# B&R Automation Studio project ABC_Pltzr (part 2)

#### bgTcpSocketClient.c
```c
/*
File: bgTcpSocketClientServer.c
=====

B&R Libraries:
==============
Make sure to add following .a files to the task using this source file:
libsys_lib.a
libbrsystem.a
libastcp.a
*/

/*
B&R components:
===============================================================================
*/
#include <bur/plc.h>
#include <bur/plctypes.h>
#include <ethsock.h>
#include <astcp.h>
#include <brsystem.h>
#include <sys_lib.h>

/*
BG components
===============================================================================
*/
#include "bgdebug.h"
#include "bgstring.h"

#include "bgTcpSocketClientServer.h"
#include "bgHttpProtocol.h"

/*
Tcp Socket Client
*/
static void bgTcpSocketClientDefaultSessionHandler(bgTcpSocketSession_typ* pSession);
static void bgTcpSocketClientSessionStateMachine(bgTcpSocketSession_typ* pSession);
static void	bgTcpSocketClientExecuteSessionHandler(bgTcpSocketSession_typ* pSession, int init);

static void bgTcpSocketClientMemAlloc(bgTcpSocketClient_typ* pClient);
static void bgTcpSocketClientSessionStart(bgTcpSocketClient_typ* pClient);
static void	bgTcpSocketClientExecuteSessionHandler(bgTcpSocketSession_typ* pSession, int init);
static void bgTcpSocketClientSessionCyclic(bgTcpSocketClient_typ* pClient);
static void bgTcpSocketClientSessionLauncher(bgTcpSocketClient_typ* pClient);
static void setSocketAddressData(ETH_sockaddr_typ *adrData, char *hostIpAddressString, unsigned short hostPort);
static void swapBytesInShort(unsigned short *value);

/*
TCP Socket Client
######################################################################################################
######################################################################################################
######################################################################################################
######################################################################################################
*/
void bgTcpSocketClientInit(bgTcpSocketClient_typ* pClient,
    int sessionSendBufSize,
    int sessionRecvBufSize,
    int applicationBufSize,
    char* pRecvBuf,
    void (*pSessionHandler)(bgTcpSocketSession_typ*),
    void (*pApplicationHandler)(bgTcpSocketSession_typ*))
{
    pClient->serverPort = 0;

	pClient->recvBuffer = pRecvBuf;

	/*Recv buffer can't be allocated! recv DOES NOT WORK if the buffer is not in PV space!?!?!?!?*/
	if(!pRecvBuf){
		DBGCRT("bgTcpSocketClientInit: recvBuf not defined!\r\n");
		pClient->memAllocStatus2 = 1;
		return;
	}

    pClient->serverIpAddr[0] = 0;

    pClient->numSupportedSessions = 1;

    pClient->sessionSendBufSize = sessionSendBufSize;

    pClient->sessionRecvBufSize = sessionRecvBufSize;

	pClient->applicationBufSize = applicationBufSize;

	/*Recv buffer can't be allocated! recv DOES NOT WORK if the buffer is not in PV space!?!?!?!?*/
    pClient->sessionTotalBufSize = pClient->sessionSendBufSize + pClient->applicationBufSize;

    pClient->totalBufSize = pClient->sessionTotalBufSize * pClient->numSupportedSessions;

    pClient->pSessionHandler = pSessionHandler;

    pClient->pApplicationHandler = pApplicationHandler;

	pClient->sockStateData = BGTCPSOCK_STATE_NONE;

	pClient->dbgDumpSendBuf = 0;
	pClient->dbgDumpRecvBuf = 0;

	/*allocate memory for send/recv buffers*/
	bgTcpSocketClientMemAlloc(pClient);

	if(pClient->memAllocStatus2 ){
			DBGCRT("bgTcpSocketClientInit: memory error! memAllocStatus2=%d\r\n", pClient->memAllocStatus2);
	}
}

void bgTcpSocketClientCyclic(bgTcpSocketClient_typ* pClient)
{
int ret;
	/*non-blocking I/O control*/
static ETH_fd_set_typ fdR;
static ETH_fd_set_typ fdW;
static ETH_timeval_typ timeOut;

	/*if memalloc fails, can't do much!*/
	if(pClient->memAllocStatus2)
		return;

	/*monitor upper layer requests to start a client session*/
	bgTcpSocketClientSessionLauncher(pClient);

	/*execute session state machine*/
	bgTcpSocketClientSessionCyclic(pClient);

	/*client state machine*/
	switch(pClient->sockStateData){
		case BGTCPSOCK_STATE_NONE:
    		return;
		break;

		case BGTCPSOCK_STATE_INITOPEN:

 			/*create socket*/
			pClient->tcpOpen.ident = socket(ETH_AF_INET, ETH_SOCK_STREAM, 0);

			if( pClient->tcpOpen.ident == ERR_SOCKET ){
				DBGMSG("socket create error (init open); EthGetError=%d\r\n", EthGetError());
				pClient->sockStateData = BGTCPSOCK_STATE_NONE;
				break;
			}

			pClient->tcpClient.ident = pClient->tcpOpen.ident;
			pClient->tcpClose.ident = pClient->tcpOpen.ident;

			/*set non-blocking socket operation*/
			{
				UDINT arg = 1;
				ioctl(pClient->tcpOpen.ident, ETH_FIONBIO, (UDINT)&arg);
			}

#if 0
			/*get sock options*/
			{
				ret = getsockopt(pClient->tcpOpen.ident, ETH_SOL_SOCKET, ETH_SO_SNDTIMEO, (UDINT)&opt1, (UDINT)&opt1size);
				DBGMSG("getsockopt ret=%d\r\n", ret);
			}
#endif

			/*reset select flags*/
			fd_zero((UDINT)&fdR);
			fd_zero((UDINT)&fdW);

			/*set time-out to 10ms*/
			timeOut.tv_sec = 0;
			timeOut.tv_usec = 1000 * 10;

			pClient->sockStateData = BGTCPSOCK_STATE_OPEN;

		case BGTCPSOCK_STATE_OPEN:

			/*connect to remote host*/
			{
			ETH_sockaddr_typ serverAdr;
			setSocketAddressData(&serverAdr, pClient->serverIpAddr, pClient->serverPort);
			ret = connect(pClient->tcpOpen.ident, (UDINT)&serverAdr, sizeof(ETH_sockaddr_typ) );
			}

			if(ret == ERR_SOCKET){
				UINT errCode = EthGetError();
				if(errCode == ERR_ETH_INPROGRESS){
					/*next: wait connect to complete*/
					DBGMSG("socket connect - wait connect to complete!\r\n");
					pClient->sockStateData = BGTCPSOCK_STATE_CLIENT;
				    break;
				}else
				if(errCode == ERR_ETH_ISCONN){
					/*it's connected -> done*/
					DBGMSG("socket connect ok(1)!\r\n");
	                bgTcpSocketClientSessionStart(pClient);
					pClient->sockStateData = BGTCPSOCK_STATE_CONNECTED;
					break;
				}
				else{
					DBGMSG("socket connect error(open); EthGetError=%d\r\n", EthGetError());
					pClient->sockStateData = BGTCPSOCK_STATE_NONE;
					break;
				}
			}
			/*connected!*/
			/*it's connected -> done*/
			DBGMSG("socket connect ok(2)!\r\n");
            bgTcpSocketClientSessionStart(pClient);
			pClient->sockStateData = BGTCPSOCK_STATE_CONNECTED;
		break;
		case BGTCPSOCK_STATE_CLIENT:
			/*select waits for connection to complete*/
			fd_set(pClient->tcpOpen.ident, (UDINT)&fdR);
			fd_set(pClient->tcpOpen.ident, (UDINT)&fdW);
			ret = sock_select(32, (UDINT)&fdR, (UDINT)&fdW, 0L, (UDINT)&timeOut);

			if(ret == ERR_SOCKET){
				DBGMSG("socket connect error; (cli) EthGetError=%d\r\n", EthGetError());
				pClient->sockStateData = BGTCPSOCK_STATE_CLOSE;
				break;
			}

			if(ret == 0){

			}else{
				if( fd_isset(pClient->tcpOpen.ident, (UDINT)&fdW) ){
					DBGMSG("socket connect(long) ok!\r\n");
	                bgTcpSocketClientSessionStart(pClient);
					pClient->sockStateData = BGTCPSOCK_STATE_CONNECTED;
				}
			}
		break;
        case BGTCPSOCK_STATE_CONNECTED:
			/*Monitor session operation; generate OnResponseReady & OnResponseError triggers*/
            /*TODO: implement timeout here -> kill sessions if stuck*/
			if(pClient->session[0].socketState == BGTCPSOCK_SESSION_STATE_NONE){
				pClient->sockStateData = BGTCPSOCK_STATE_NONE;
			}
        break;
        case BGTCPSOCK_STATE_CLOSE:
			close(pClient->tcpClose.ident);
	    	pClient->sockStateData = BGTCPSOCK_STATE_NONE;
			DBGMSG("bgTcpSocketClientSessionStateMachine(): closing socket\r\n");
        break;
        case BGTCPSOCK_STATE_ERROR:
        break;
	 }

    return;
}

static void bgTcpSocketClientMemAlloc(bgTcpSocketClient_typ* pClient)
{
unsigned int memSize;
int i;

	/*Get System Memory Information*/
	pClient->MEMInfo.enable = 1;
	MEMInfo(&pClient->MEMInfo);

	memSize = pClient->totalBufSize;

	/*allocate space for send/recv buffers*/
	if(pClient->sendRecvBuffer == 0){
		/* allocate new memory from RAM*/
    	pClient->memAllocStatus2 = TMP_alloc(memSize, (void**)&pClient->sendRecvBuffer);
	}else{
		/*memory is allready allocated -> free it first!*/
    	pClient->memAllocStatus2 = TMP_free(memSize, (void**)pClient->sendRecvBuffer);

    	/*allocate new memory from RAM*/
    	pClient->memAllocStatus2 = TMP_alloc(memSize, (void**)pClient->sendRecvBuffer);
	}

	/*assign send/recv buffer ptrs*/
    pClient->session[0].pSendBuf = (char*)(pClient->sendRecvBuffer + i * pClient->sessionTotalBufSize);
	pClient->session[0].sendBufLength = pClient->sessionSendBufSize;

    pClient->session[0].pAppBuf = (char*)(pClient->session[0].pSendBuf + pClient->sessionSendBufSize);
	pClient->session[0].appBufLength = pClient->applicationBufSize;

    pClient->session[0].pRecvBuf = pClient->recvBuffer;
	pClient->session[0].recvBufLength = pClient->sessionRecvBufSize;
}

static void bgTcpSocketClientSessionStart(bgTcpSocketClient_typ* pClient)
{
int i;
bgTcpSocketSession_typ *pSession;

	/* client: pClient->numSupportedSessions = 1 ALWAYS!*/
    for(i=0; i < pClient->numSupportedSessions; i++){
        if( pClient->session[i].socketState == BGTCPSOCK_SESSION_STATE_NONE){
            pSession = &pClient->session[i];
            pSession->socketState = BGTCPSOCK_SESSION_STATE_SEND;

			pSession->tcpSend.enable = 1;
			pSession->tcpSend.ident = pClient->tcpOpen.ident;   		/* copy the  Ident number */
			pSession->tcpSend.flags = 0;
			pSession->tcpSend.pData = (UDINT)pSession->pSendBuf;

			pSession->tcpRecv.enable = 1;
			pSession->tcpRecv.ident = pClient->tcpOpen.ident;     		/* copy the  Ident number */

			pSession->tcpRecv.pData = (UDINT)pSession->pRecvBuf;        /* address of the buffer */;

			pSession->tcpRecv.datamax = pClient->sessionRecvBufSize;    /* length of the buffer */;

			pSession->tcpClose.enable = 1;
   			pSession->tcpClose.ident = pClient->tcpOpen.ident;    		/* copy the  Ident number */

			pSession->pTcpLayer = (char*)pClient;	                    /*session has ptr to tcp layer*/

            pSession->rxByteCount = 0;
            brsstrcpy((UDINT)pSession->clientIpAddr, (UDINT)pClient->clientIpAddr);

			pSession->dbgDumpRecvBuf = pClient->dbgDumpRecvBuf;
			pSession->dbgDumpSendBuf = pClient->dbgDumpSendBuf;

			/*init session specific handler - call the handler with init pSession->flag=1*/
			bgTcpSocketClientExecuteSessionHandler(pSession, 1);

			DBGMSG("bgTcpSocketClientSessionStart(): connection to %s, starting session Id= %d\r\n", pClient->serverIpAddr, i);
            return;
        }
    }

	DBGCRT("bgTcpSocketClientSessionStart(): client busy! activeSessions= %d\r\n", pClient->numSupportedSessions);
    pClient->sockStateData = BGTCPSOCK_STATE_TOOBUSY;
}

static void	bgTcpSocketClientExecuteSessionHandler(bgTcpSocketSession_typ* pSession, int init)
{
bgTcpSocketClient_typ* pClient = (bgTcpSocketClient_typ*)pSession->pTcpLayer;

	pSession->init = 0;
	if( init )
		pSession->init = 1;

	DBGMSG("bgTcpSocketClientExecuteSessionHandler\r\n p1=%d p2=%d\r\n", pClient->pSessionHandler, bgHttpClientSessionHandler);

/*
	bgHttpClientSessionHandler(pSession);
*/
    if(pClient->pSessionHandler)
    	(*pClient->pSessionHandler)(pSession);
    else
    	bgTcpSocketClientDefaultSessionHandler(pSession);

	pSession->init = 0;
}

static void bgTcpSocketClientSessionCyclic(bgTcpSocketClient_typ* pClient)
{
int i;
bgTcpSocketSession_typ *pSession;
int activeSessions = 0;

    for(i=0; i < pClient->numSupportedSessions; i++){
        pSession = &pClient->session[i];

        if( pSession->socketState != BGTCPSOCK_SESSION_STATE_NONE){
            activeSessions++;
            bgTcpSocketClientSessionStateMachine(pSession);
        }
    }
    pClient->numActiveSessions = activeSessions;
}

static void bgTcpSocketClientSessionLauncher(bgTcpSocketClient_typ* pClient)
{
int i;
bgTcpSocketSession_typ *pSession;

    for(i=0; i < pClient->numSupportedSessions; i++){
        pSession = &pClient->session[i];

		if( (pSession->bSendData) ){
			pSession->bSendData = 0;
			if(pClient->sockStateData == BGTCPSOCK_STATE_NONE){
				pClient->sockStateData = BGTCPSOCK_STATE_INITOPEN;
			}else{
				DBGMSG("bgTcpSocketClientSessionLauncher: client session start rejected; client is busy! cliState=%d\r\n",
					pClient->sockStateData);
			}
		}
    }
}
static void bgTcpSocketClientSessionStateMachine(bgTcpSocketSession_typ* pSession)
{
int ret;

    switch(pSession->socketState){
		case BGTCPSOCK_SESSION_STATE_SEND:

        	ret = send(pSession->tcpSend.ident, (UDINT)pSession->pSendBuf, pSession->tcpSend.datalen, 0L);

        	if(ret == ERR_SOCKET){
				DBGMSG("send error EthGetError=%d\r\n", EthGetError());
				pSession->socketState = BGTCPSOCK_SESSION_STATE_CLOSE;    /*close this socket*/
				return;
        	}

			/*remember the send length*/
			DBG("send() ok; bytes=%d\r\n", (int)ret);
			pSession->tcpSend.sentlen = ret;
	   		pSession->socketState = BGTCPSOCK_SESSION_STATE_RECEIVE;    /*close this socket session*/

		/*break;*/

		case BGTCPSOCK_SESSION_STATE_RECEIVE:
	       	/*call receive (NON BLOCKING MODE!)*/
        	ret = recv(pSession->tcpRecv.ident, (UDINT)pSession->tcpRecv.pData, pSession->tcpRecv.datamax, 0L);

        	if(ret == ERR_SOCKET){
        		UINT errCode = EthGetError();
        		/*none blocking receive return this following value if data is not available yet*/
        		if( errCode == ERR_ETH_WOULDBLOCK ){
        			/*wait response*/
					return;
        		}
				DBGMSG("RxError EthGetError=%d\r\n", errCode);
	   			pSession->socketState = BGTCPSOCK_SESSION_STATE_CLOSE;    /*close this socket session*/
				break;
        	}

			pSession->tcpRecv.recvlen = ret;

            if(pSession->tcpRecv.recvlen){
				DBGMSG("rx OK! rxLen=%d\r\n", ret);

				bgTcpSocketClientExecuteSessionHandler(pSession, 0);

				/*uper layer completed processing? */
				if( pSession->bCloseSession){
					pSession->bCloseSession = 0;
	   					pSession->socketState = BGTCPSOCK_SESSION_STATE_CLOSE;    /*close this socket session*/
				}
            }else{
				DBGMSG("bgTcpSocketClient..: RMT SOCK CLOSED!\r\n");
	   			pSession->socketState = BGTCPSOCK_SESSION_STATE_CLOSE;    /*close this socket session*/
			}
			return;
		break;

		case BGTCPSOCK_SESSION_STATE_CLOSE:
			close(pSession->tcpClose.ident);
	    	pSession->socketState = BGTCPSOCK_SESSION_STATE_NONE;
			DBGMSG("bgTcpSocketClientSessionStateMachine(): stopping session Id= %d\r\n", pSession->ident);
		break;

		case BGTCPSOCK_SESSION_STATE_DELAY:
			pSession->delayCounter--;
			if(pSession->delayCounter <= 0)
    			pSession->socketState = BGTCPSOCK_SESSION_STATE_CLOSE;    /*close this server socket*/
		break;

		default:

		break;
	}
}

#if 0
static void bgTcpSocketClientSessionSendData(bgTcpSocketSession_typ* pSession, int len)
{
	pSession->tcpSend.datalen = len;
	pSession->socketState = BGTCPSOCK_STATE_INITOPEN;

#if 0
{
int i;
char text[90];
/*session/application/protocol specific data structure*/
httpRequest_typ* r = (httpRequest_typ*)pSession->pProtocol;

	DBGMSG("bgHttpSend(): lenght(bytes): total=%d(%d) header=%d content=%d\r\n",
		len, r->sendTotalLength, r->sendHeaderLength, r->sendContentLength);

	DBGMSG("bgHttpSend dump:\r\n");
	DBGMSG("============================================\r\n");
	for(i=0;i<len; i++){
 		if( ((i+1)*80) < len ){
			memcpy(&text[0], &pSession->pSendBuf[i*80], 80);
			text[80]=0;
			DBGMSG("%s", &text[0]);
		}else{
			memcpy(&text[0], &pSession->pSendBuf[i*80], len - (i*80));
			text[len - (i*80)]=0;
			DBGMSG("%s", &text[0]);
			break;
		}
	}
	DBGMSG("============================================\r\n\r\n");
}
#endif

}
#endif
/*
Default session handler
######################################################################################################
######################################################################################################
######################################################################################################
######################################################################################################
*/
static void bgTcpSocketClientDefaultSessionHandler(bgTcpSocketSession_typ* pSession)
{
    /*default session handler -> send out http error response "internal server error"*/
/*    httpSendErrorResponse(pSession, 500);
*/
}

static void setSocketAddressData(ETH_sockaddr_typ *adrData, char *hostIpAddressString, unsigned short hostPort)
{

	unsigned short sin_family;
	unsigned short family;
	unsigned short length;
	unsigned short port;

	family = ETH_AF_INET;
	length = sizeof(ETH_sockaddr_typ);
	sin_family = (family << 8) + length;

	adrData->sin_family = sin_family;
	port = hostPort;
	swapBytesInShort(&port);
	adrData->sin_port = port;
	if( strlen(hostIpAddressString) < 8)
		adrData->sin_addr = ETH_INADDR_ANY;
	else
		adrData->sin_addr = inet_addr( (unsigned long) hostIpAddressString);
	adrData->sin_zero[0]=0;
	adrData->sin_zero[1]=0;
	adrData->sin_zero[2]=0;
	adrData->sin_zero[3]=0;
	adrData->sin_zero[4]=0;
	adrData->sin_zero[5]=0;
	adrData->sin_zero[6]=0;
	adrData->sin_zero[7]=0;
}

static void swapBytesInShort(unsigned short *value)
{

union{
	unsigned short 	shortValue;
	unsigned char	bytes[2];
}swapValue;

unsigned char tempByte;

	swapValue.shortValue = *value;
	tempByte = swapValue.bytes[0];
	swapValue.bytes[0] = swapValue.bytes[1];
	swapValue.bytes[1] = tempByte;
	*value = swapValue.shortValue;
}
```

### paiFileService.typ
```iecst
(********************************************************************
 * COPYRIGHT --
 ********************************************************************
 * Package: paiFileService
 * File: paiFileService.typ
 * Author: goran_2
 * Created: August 05, 2011
 ********************************************************************
 * Data types of package paiFileService
 ********************************************************************)

TYPE
	PAI_FILESERVICE_ENUMS :
		(
		PAI_FS_DEVICE_MAXIDX := 19,
		PAI_FS_DEVICE_NONE := 0,
		PAI_FS_IDLE := 0,
		PAI_FS_RDFILE := 1,
		PAI_FS_WRFILE := 2,
		PAI_FS_INFOFILE := 3,
		PAI_FS_DELFILE := 4,
		PAI_FS_RDDIR := 10,
		PAI_FS_CRDIR := 11,
		PAI_FS_INFODIR := 12
		);
	paiFileServiceDevDirItem_typ : 	STRUCT
		deviceName : STRING[31];
		dirName : STRING[127];
		deviceConfiguration : STRING[127];
		createdAtPowerUp : BOOL;
		status : INT;
	END_STRUCT;
	paiFileServiceDeviceTable_typ : 	STRUCT
		listDevsDirs : ARRAY[0..19]OF paiFileServiceDevDirItem_typ;
	END_STRUCT;
	paiFileServicePublicIn_typ : 	STRUCT
		request : USINT;
		adrDeviceName : UDINT; (*Address of the Device Name*)
		adrName : UDINT; (*File/dir name for the requested action (read, write, create, delete, etc)*)
		adrName2 : UDINT; (*File/dir name for the requested action (read, write, create, delete, etc)*)
		adrReadDst : UDINT; (*Destination address for the read action*)
		readDstLen : UDINT; (*Length of the space available for read at the given address*)
		readOffset : UDINT;
		adrWriteSrc : UDINT; (*Src address for the write action.*)
		writeSrcLen : UDINT; (*Length of data available at src address*)
		writeOffset : UDINT;
		pCallback : UDINT; (*ptr to Callback function*)
		pCallbackData : UDINT; (*ptr to Callback data*)
	END_STRUCT;
	paiFileServicePublicOut_typ : 	STRUCT
		status : UINT; (*Output status for R or W request. Valid when writeDone or readDone set to 1.*)
		initOk : BOOL; (*Output status that indicates if service completed initialization after system start. Wait with any access until initOk == 1*)
		busy : BOOL; (*Output status to indicate that service is busy (busy == 1) servicing a current request. Avoid issuing new requests.*)
		powerUp : BOOL; (*Output status to indicate that service completed servicing a current request. Shall be cleared by the receiver of the event.*)
		done : BOOL; (*Output status to indicate that service completed servicing a current request. Shall be cleared by the receiver of the event.*)
		bytecount : UDINT; (*Number of bytes during file read.*)
	END_STRUCT;
	paiFileServicePrivateFileFBK_typ : 	STRUCT
		open : FileOpen;
		close : FileClose;
		read : FileRead;
		readex : FileReadEx;
		write : FileWrite;
		writeex : FileWriteEx;
		copy : FileCopy;
		create : FileCreate;
		delete : FileDelete;
		rename : FileRename;
		truncate : FileTruncate;
		info : FileInfo;
		infoData : fiFILE_INFO;
	END_STRUCT;
	paiFileServicePrivateDevFBK_typ : 	STRUCT
		link : DevLink;
		unlink : DevUnlink;
	END_STRUCT;
	paiFileServiceDirFBK_typ : 	STRUCT
		open : DirOpen;
		close : DirClose;
		read : DirRead;
		copy : DirCopy;
		create : DirCreate;
		delete : DirDelete;
		deleteex : DirDeleteEx;
		rename : DirRename;
		info : DirInfo;
	END_STRUCT;
	paiFileServicePrivate_typ : 	STRUCT
		requestType : USINT;
		status : UINT;
		bgssm : bgSSM_typ;
		currentDeviceIndex : UDINT;
		pDeviceTable : REFERENCE TO paiFileServiceDeviceTable_typ;
		device : paiFileServicePrivateDevFBK_typ;
		dir : paiFileServiceDirFBK_typ;
		file : paiFileServicePrivateFileFBK_typ;
	END_STRUCT;
	paiFileService_typ : 	STRUCT
		i : paiFileServicePublicIn_typ;
		o : paiFileServicePublicOut_typ;
		prv : paiFileServicePrivate_typ;
	END_STRUCT;
END_TYPE
```

### Program Logical/paiComponents/paiFileService/paiFS (ANSIC)

#### paiDevDirConfigure.c - pai FS Device and Directory configuration
```c
/********************************************************************
 * COPYRIGHT --
 ********************************************************************
 * Program: paiFile
 * File: paiDevDirConfigure.c
 * Author: goran_2
 * Created: August 05, 2011
 ********************************************************************
 * Implementation of program paiDevDirConfigure
 ********************************************************************/

#include <bur/plctypes.h>

#ifdef _DEFAULT_INCLUDES
 #include <AsDefault.h>
#endif

#include "paiFile.h"

/*
###############################################################################
PAI_CONFIGURATION_SECTION
Code below allows configuration of the devices and folders used in the
application.
###############################################################################
*/
#warning "pai Configuration: application File Devices and Folders"
void paiFSDeviceAndDirConfig( void )
{
	int idx=0;
	//If .deviceConfiguration is NOT empty string, entry is related to device link at powerup
	//If .deviceConfiguration is empty string, entry is related to directory check/create at powerup

	brsstrcpy((UDINT)paiFSDevices.listDevsDirs[idx].deviceName, (UDINT)PAI_FS_DEVICE_ROOT);
	brsstrcpy((UDINT)paiFSDevices.listDevsDirs[idx].dirName, (UDINT)"");
	brsstrcpy((UDINT)paiFSDevices.listDevsDirs[idx].deviceConfiguration, (UDINT)PAI_FS_DEVICE_ROOT_CFG);

	idx++;
	brsstrcpy((UDINT)paiFSDevices.listDevsDirs[idx].deviceName, (UDINT)PAI_FS_DEVICE_ROOT);
	brsstrcpy((UDINT)paiFSDevices.listDevsDirs[idx].dirName, (UDINT)PAI_FS_APP_DIR_DATA);//i.e. Data
	brsstrcpy((UDINT)paiFSDevices.listDevsDirs[idx].deviceConfiguration, (UDINT)"");

	idx++;
	brsstrcpy((UDINT)paiFSDevices.listDevsDirs[idx].deviceName, (UDINT)PAI_FS_DEVICE_ROOT);
	brsstrcpy((UDINT)paiFSDevices.listDevsDirs[idx].dirName, (UDINT)PAI_FS_APP_DIR_CFG);//i.e. Data/Cfg
	brsstrcpy((UDINT)paiFSDevices.listDevsDirs[idx].deviceConfiguration, (UDINT)"");

	idx++;
	brsstrcpy((UDINT)paiFSDevices.listDevsDirs[idx].deviceName, (UDINT)PAI_FS_DEVICE_ROOT);
	brsstrcpy((UDINT)paiFSDevices.listDevsDirs[idx].dirName, (UDINT)PAI_FS_APP_DIR_REC);//i.e. Data/Rec
	brsstrcpy((UDINT)paiFSDevices.listDevsDirs[idx].deviceConfiguration, (UDINT)"");

	idx++;
	brsstrcpy((UDINT)paiFSDevices.listDevsDirs[idx].deviceName, (UDINT)PAI_FS_DEVICE_ROOT);
	brsstrcpy((UDINT)paiFSDevices.listDevsDirs[idx].dirName, (UDINT)"Data/Rec/Layers");//i.e. Data/Rec/Layers
	brsstrcpy((UDINT)paiFSDevices.listDevsDirs[idx].deviceConfiguration, (UDINT)"");

	idx++;
	brsstrcpy((UDINT)paiFSDevices.listDevsDirs[idx].deviceName, (UDINT)PAI_FS_DEVICE_ROOT);
	brsstrcpy((UDINT)paiFSDevices.listDevsDirs[idx].dirName, (UDINT)"Data/Rec/Pallets");//i.e. Data/Rec/Pallets
	brsstrcpy((UDINT)paiFSDevices.listDevsDirs[idx].deviceConfiguration, (UDINT)"");

	idx++;
	brsstrcpy((UDINT)paiFSDevices.listDevsDirs[idx].deviceName, (UDINT)PAI_FS_DEVICE_ROOT);
	brsstrcpy((UDINT)paiFSDevices.listDevsDirs[idx].dirName, (UDINT)"Data/Test");
	brsstrcpy((UDINT)paiFSDevices.listDevsDirs[idx].deviceConfiguration, (UDINT)"");

	idx++;
	brsstrcpy((UDINT)paiFSDevices.listDevsDirs[idx].deviceName, (UDINT)PAI_FS_DEVICE_CFG);
	brsstrcpy((UDINT)paiFSDevices.listDevsDirs[idx].dirName, (UDINT)"");
	brsstrcpy((UDINT)paiFSDevices.listDevsDirs[idx].deviceConfiguration, (UDINT)PAI_FS_DEVICE_CFG_CFG);

	idx++;
	brsstrcpy((UDINT)paiFSDevices.listDevsDirs[idx].deviceName, (UDINT)PAI_FS_DEVICE_REC);
	brsstrcpy((UDINT)paiFSDevices.listDevsDirs[idx].dirName, (UDINT)"");
	brsstrcpy((UDINT)paiFSDevices.listDevsDirs[idx].deviceConfiguration, (UDINT)PAI_FS_DEVICE_REC_CFG);

	idx++;
	brsstrcpy((UDINT)paiFSDevices.listDevsDirs[idx].deviceName, (UDINT)PAI_FS_DEVICE_REC_LAYER);
	brsstrcpy((UDINT)paiFSDevices.listDevsDirs[idx].dirName, (UDINT)"");
	brsstrcpy((UDINT)paiFSDevices.listDevsDirs[idx].deviceConfiguration, (UDINT)PAI_FS_DEVICE_REC_LAYER_CFG);

	idx++;
	brsstrcpy((UDINT)paiFSDevices.listDevsDirs[idx].deviceName, (UDINT)PAI_FS_DEVICE_REC_PALLETE);
	brsstrcpy((UDINT)paiFSDevices.listDevsDirs[idx].dirName, (UDINT)"");
	brsstrcpy((UDINT)paiFSDevices.listDevsDirs[idx].deviceConfiguration, (UDINT)PAI_FS_DEVICE_REC_PALLETE_CFG);

	idx++;
	brsstrcpy((UDINT)paiFSDevices.listDevsDirs[idx].deviceName, (UDINT)"USB1");
	brsstrcpy((UDINT)paiFSDevices.listDevsDirs[idx].dirName, (UDINT)"");
	brsstrcpy((UDINT)paiFSDevices.listDevsDirs[idx].deviceConfiguration, (UDINT)"/DEVICE=IF3.ST1");

	idx++;
	brsstrcpy((UDINT)paiFSDevices.listDevsDirs[idx].deviceName, (UDINT)"USB2");
	brsstrcpy((UDINT)paiFSDevices.listDevsDirs[idx].dirName, (UDINT)"");
	brsstrcpy((UDINT)paiFSDevices.listDevsDirs[idx].deviceConfiguration, (UDINT)"/DEVICE=IF4.ST1");

}
//eof
```

### Program Logical/paiComponents/paiHmi

#### paiHmiSystemDateTime.h
```c
/********************************************************************
 * COPYRIGHT -- pai
 ********************************************************************
 * Program: hmilogic
 * File: hmiAlert.h
 * Author: goran
 * Created: September 05, 2013
 *******************************************************************/

#include <bur/plctypes.h>
#ifdef _DEFAULT_INCLUDES
#include <AsDefault.h>
#endif
void paiHmiSystemDateTimeInit(paiHmiSystemTime_typ* p);
void paiHmiSystemDateTimeCyclic(paiHmiSystemTime_typ* p);
```

#### paiHmiTableViewProducts.c
```c
/********************************************************************
 * COPYRIGHT -- pai
 ********************************************************************
 * Program: hmilogic
 * File: hmiTableViewPersons.c
 * Author: goran
 * Created: November 24, 2013
 ********************************************************************
 * Implementation of program hmiTableViewProducts
 ********************************************************************/

#include <bur/plctypes.h>

#ifdef _DEFAULT_INCLUDES
	#include <AsDefault.h>
#endif

/**
Bit manipulaiton utility functions.
 */
//#include <../../bglib/bgBitUtilities.h>

/**
String manipulaiton utility functions.
 */
#include <../../bglib/bgsprintf.h>
//#include <../../bglib/bgstring.h>

//#include <../../RecFIFO/fifotest/fifoif.h>
/*
###############################################################################
Table View support functions
###############################################################################
*/

/*
Display table background grid (i.e. each odd row in one color, each even row in
a different color
*/
void tableViewShowGridProducts(hmiTableProducts_typ* p)
{
	int ii;

	for(ii=0; ii<=p->viewIndexMax; ii++){
		//select a different collor scheme for each row of the table
		if(ii%2){
			p->itemsInView[ii].ctrl.bgdColorIndex = 1;
		}else{
			p->itemsInView[ii].ctrl.bgdColorIndex = 0;
		}
	}
}

void tableFilterExecuteProducts(hmiTableProducts_typ* p)
{
	if(!p)
		return;

	p->executeFilter = 1;//execute filter request; cleared upon filter execution
}
static int tableFilterIsUpdateProducts(hmiTableProducts_typ* p, int* filterType)
{
	int filterLocal = 0;
	int filterDB = 0;

	if(!p){
		if(filterType)
			*filterType = 0;
		return 0;
	}

	//filter setting changed?
	if( !p->executeFilter &&
		(p->shiftFilter == p->shiftFilterOld) &&
		(p->activeFilter == p->activeFilterOld) &&
		(p->assignedFilter == p->assignedFilterOld) &&
		(p->azFilterFirstName == p->azFilterFirstNameOld) &&
		(p->azFilterLastName == p->azFilterLastNameOld)
	){
		//no changes for filters that required DB request
	}else{
		filterDB = 1;
	}

	if( (p->assignedFilter == p->assignedFilterOld) ){
		//no changes for filters that are performed localy
	}else{
		filterLocal = 1;
	}

	p->executeFilter = 0;
	p->shiftFilterOld = p->shiftFilter;
	p->activeFilterOld = p->activeFilter;
	p->assignedFilterOld = p->assignedFilter;
	p->azFilterLastNameOld = p->azFilterLastName;
	p->azFilterFirstNameOld = p->azFilterFirstName;

	*filterType = filterDB + (2 * filterLocal);//bit0-filterDB, bit1-filterLocal

	return 1;
}
/*
Init table based person viewer
*/
void tableViewProductsInit(hmiTableProducts_typ* p, hmiTableItemDataProduct_typ* pItemsAll, UDINT itemCount, UDINT viewIndexMax, char* pDBTableName, int jsonSQLQueryid)
{
	int ii;

	if(!p || !pItemsAll || !itemCount || !viewIndexMax)
		return;

	p->pItemsAll = (UDINT)pItemsAll;

	p->viewIndexMax = viewIndexMax;
	if(p->viewIndexMax > hmiTableProductsMAXVIEWINDEX){
		p->viewIndexMax = hmiTableProductsMAXVIEWINDEX;
	}

	tableViewShowGridProducts(p);

	//reset selection/activate indexes and datapoints wired to hotspots
	p->selectedItem = -1;
	p->selectedViewItem = -1;
	p->selectViewItemDataPoint = -1;
	p->activateViewItemDataPoint = -1;
	if(pDBTableName)
		brsstrcpy((UDINT)p->activeDBTableName, (UDINT)pDBTableName);
	p->activeSQLid = jsonSQLQueryid;

	//simulate some data
	p->itemCountUnfiltered = 0;
	p->itemCount = 0;
	for(ii=0; ii<itemCount;ii++){
		if(pItemsAll[ii].usedEntry){
			p->itemCountUnfiltered++;
			p->itemCount++;
		}
	}
}

/*
Hide (don't show) table row data at a selected row. Result is an empty line.
*/
static void productTableHideItemAtIndex(hmiTableProducts_typ* p, int viewIndex)
{
	if(!p || viewIndex > p->viewIndexMax)
		return;
	p->itemsInView[viewIndex].ctrl.visibilityControl = 1;
}

/*
Show (don't hide) table row data at a selected row. Result is an line that contais all columns (i.e. text fields).
*/
static void productTableShowItemAtIndex(hmiTableProducts_typ* p, int viewIndex)
{
	if(!p || viewIndex > p->viewIndexMax)
		return;

	//convert numerics into txt
	//bgsprintf(p->itemsInView[viewIndex].data.employeeIdTxt, "%d", p->itemsInView[viewIndex].data.employeeId);
	bgsprintf(p->itemsInView[viewIndex].data.indexTxt, "%d", p->itemsInView[viewIndex].data.index);
	//bgsprintf(p->itemsInView[viewIndex].data.shiftTxt, "%d", p->itemsInView[viewIndex].data.shift);

	//make item visible
	p->itemsInView[viewIndex].ctrl.visibilityControl = 0;
}

/*
Display table view.
*/
void tableViewShowProducts(hmiTableProducts_typ* p)
{
	int ii, jj;
	hmiTableItemDataProduct_typ* pItemsAll;

	if(!p || !p->pItemsAll)
		return;

	pItemsAll = (hmiTableItemDataProduct_typ*)p->pItemsAll;

	for(ii=0, jj = p->viewIndex; ii<=p->viewIndexMax; jj++){
		if(pItemsAll[jj].index < 0)
			continue;

		if(jj<p->itemCountUnfiltered){
			brsmemcpy((UDINT)&p->itemsInView[ii].data, (UDINT)&pItemsAll[jj], sizeof(hmiTableItemDataProduct_typ) );
			productTableShowItemAtIndex(p, ii);
		}else{
			productTableHideItemAtIndex(p, ii);
		}
		ii++;
	}
}

/*
Selection (i.e. row highlighting) of the table row.
*/
static void tableViewItemSelectionProducts(hmiTableProducts_typ* p)
{
	if(!p)
		return;

	//table item selection logic
	//selectViewItemDataPoint is connected to a hotstop above the table line. Each line sets a different
	//number that corepsonds to the visible (table) line number.
	if( (p->selectViewItemDataPoint >= 0) && (p->selectViewItemDataPoint <= p->viewIndexMax)){
		//check if a table line is already selected
		if(p->selectedViewItem < 0){
			//no item selected > select it now
			p->selectedViewItem = p->selectViewItemDataPoint; //save selected line for lated
			p->bgdColorIndexOldSelection = p->itemsInView[p->selectedViewItem].ctrl.bgdColorIndex;//save current color index for the line to be able to restore it
			p->itemsInView[p->selectedViewItem].ctrl.bgdColorIndex = 2;//select 3-rd color from the map
			//save current selection
			p->selectedViewItem = p->selectViewItemDataPoint;
		}else
			if(p->selectedViewItem == p->selectViewItemDataPoint){
			//same item is already selected > deselect it now (toggle selection)
			//restore background color for the line
			p->itemsInView[p->selectedViewItem].ctrl.bgdColorIndex = p->bgdColorIndexOldSelection;
			//reset selection status
			p->selectedViewItem = -1;
		}else{
			//deactivate old selection, activate new selection
			p->itemsInView[p->selectedViewItem].ctrl.bgdColorIndex = p->bgdColorIndexOldSelection;
			p->bgdColorIndexOldSelection = p->itemsInView[p->selectViewItemDataPoint].ctrl.bgdColorIndex;
			p->itemsInView[p->selectViewItemDataPoint].ctrl.bgdColorIndex = 2;
			//save current selection
			p->selectedViewItem = p->selectViewItemDataPoint;
		}

		//calculate a line from the entire table that is currently selected
		p->selectedItem = -1;
		if(p->selectedViewItem >= 0)
			p->selectedItem = p->selectedViewItem + p->viewIndex;

		//reset datapoint connected to hotspots
		p->selectViewItemDataPoint = -1;
	}
}

static void tableViewRefreshProducts(hmiTableProducts_typ* p)
{
	p->selectedViewItem = -1;//invalidate view selection for a proper redraw of the selected item
	tableViewShowGridProducts(p); //redraw table layout
	tableViewShowProducts(p); //redraw table data
}

static void tableViewScrollProducts(hmiTableProducts_typ* p)
{
	if(!p || !p->itemCount)
		return;

	//if no item is selected, and any scroll key pressed, just select a top item on the list
	if( (p->selectedItem < 0) &&
		(p->btnScrollLineUp || p->btnScrollPageUp || p->btnScrollLineDw || p->btnScrollPageDw)){
		p->btnScrollLineUp = 0; p->btnScrollPageUp = 0;
		p->btnScrollLineDw = 0; p->btnScrollPageDw = 0;
		//item is NOT selected > select the top item
		p->selectViewItemDataPoint = 0;
		tableViewItemSelectionProducts(p);
		return;
	}

	//table scroll logic
	if(p->btnScrollLineUp){
		p->btnScrollLineUp = 0;

		if(!p->selectedItem){
			return;//top item is already selected > nothing to do
		}

		if(!p->selectedViewItem){
			//selected view item is at the TOP
			//is the view index > 0 (which means that scroll window has a chance to to move up)
			if(p->viewIndex){
				//view index is not all the way up > scroll it up
				p->viewIndex--;
				tableViewRefreshProducts(p);//display the entire table
			}
			p->selectViewItemDataPoint = 0;//select the top line in the view
		}else{
			//selected view item is not the TOP > need to scroll up selection within the visible view
			p->selectViewItemDataPoint = p->selectedViewItem -  1;
		}
		//update selection
		tableViewItemSelectionProducts(p);
		return;
	}

	if(p->btnScrollLineDw){
		p->btnScrollLineDw = 0;

		//item is already selected > scroll line dw
		if(p->selectedItem == (p->itemCount - 1)){
			//last item is already selected
			return;
		}

		if(p->selectedViewItem >= p->viewIndexMax){
			//selected view item is the LAST item in the view
			if(p->viewIndex < (p->itemCount - (p->viewIndexMax + 1) ) ){
				//view index can be further moved  > scroll
				p->viewIndex++;
				tableViewRefreshProducts(p);
			}
			p->selectViewItemDataPoint = p->viewIndexMax;//select last item in the table view
		}else{
			//selected view item is not the BOTTOM > scroll
			p->selectViewItemDataPoint = p->selectedViewItem +  1;
		}
		tableViewItemSelectionProducts(p);
		return;
	}

	if(p->btnScrollPageUp){
		p->btnScrollPageUp = 0;

		//is view window at the top?
		if(p->viewIndex){
			//no > scroll up by the page size
			p->viewIndex -= p->viewIndexMax+1;
			//viewIndex cann't be < 0!
			if(p->viewIndex < 0){
				p->viewIndex = 0;
				p->selectViewItemDataPoint = 0;
			}else{
				p->selectViewItemDataPoint = p->selectedViewItem;
			}
			tableViewRefreshProducts(p);//display the entire table
		}else{
			//view window is alreday all the way up > select the top line on the view
			if(p->selectedViewItem)
				p->selectViewItemDataPoint = 0;
		}
		//redraw selection
		tableViewItemSelectionProducts(p);
		return;
	}

	if(p->btnScrollPageDw){
		p->btnScrollPageDw = 0;

		//is the selection at the bottom?
		if((p->itemCount -1) <= p->selectedItem){
			//view window is alreday all the way dw > select the bottom line on the view
			return;
		}

		//no > scroll dw by the page size
		if( ((p->itemCount) / (p->viewIndexMax+1)) > ((p->selectedItem + 1) / (p->viewIndexMax+1))){
			p->viewIndex += p->viewIndexMax+1;
			if(p->viewIndex > (p->itemCount - 1 )){
				p->viewIndex = (p->itemCount - 1);
			}
			//p->selectViewItemDataPoint = p->selectedViewItem;
			p->selectViewItemDataPoint = 0;
			tableViewRefreshProducts(p);
		}

		//redraw selection
		tableViewItemSelectionProducts(p);
		return;
	}

}

/*
SELECT id,name,description,yield,pieceweight FROM products
*/
static void tableFilterProducts(hmiTableProducts_typ* p)
{
	int filterMode;//bit0-DBfilter, bit1-localFilter

	char textBuf[32];
	char gUdpClient_txbuf[768];

	if(!p || !p->pItemsAll)
		return;

	//check if running a filter is requested?
	if( !tableFilterIsUpdateProducts(p, &filterMode) )
		return ;

	if(filterMode & 0x2){
		//local filter (station assigment)
		//DBG(lgr, "Apply filter: station assing");
	}

	if(!(filterMode & 0x1)){
		return;
	}

	brsstrcpy((UDINT)&gUdpClient_txbuf[0], (UDINT)"{\"paipvilite\": \"1.0\", \"method\": \"executesqlquery\", \"params\": {\"sqlquery\":\"SELECT id,prod_name,description,yield,pieceweight,pass_score,lightFeatYieldRedPct,lightFeatYieldGreenPct,lightFeatPcPMRed,lightFeatPcPMGreen,");
	brsstrcat((UDINT)&gUdpClient_txbuf[0], (UDINT)"defect_dem_1,");
	brsstrcat((UDINT)&gUdpClient_txbuf[0], (UDINT)"defect_dem_2,");
	brsstrcat((UDINT)&gUdpClient_txbuf[0], (UDINT)"defect_dem_3,");
	brsstrcat((UDINT)&gUdpClient_txbuf[0], (UDINT)"defect_dem_4,");
	brsstrcat((UDINT)&gUdpClient_txbuf[0], (UDINT)"defect_dem_5,");
	brsstrcat((UDINT)&gUdpClient_txbuf[0], (UDINT)"defect_dem_6,");
	brsstrcat((UDINT)&gUdpClient_txbuf[0], (UDINT)"defect_dem_7,");
	brsstrcat((UDINT)&gUdpClient_txbuf[0], (UDINT)"defect_dem_8,");
	brsstrcat((UDINT)&gUdpClient_txbuf[0], (UDINT)"defect_dem_9,");
	brsstrcat((UDINT)&gUdpClient_txbuf[0], (UDINT)"defect_dem_10,");
	brsstrcat((UDINT)&gUdpClient_txbuf[0], (UDINT)"defect_dem_11,");
	brsstrcat((UDINT)&gUdpClient_txbuf[0], (UDINT)"defect_dem_12,");
	brsstrcat((UDINT)&gUdpClient_txbuf[0], (UDINT)"defect_desc_1,");
	brsstrcat((UDINT)&gUdpClient_txbuf[0], (UDINT)"defect_desc_2,");
	brsstrcat((UDINT)&gUdpClient_txbuf[0], (UDINT)"defect_desc_3,");
	brsstrcat((UDINT)&gUdpClient_txbuf[0], (UDINT)"defect_desc_4,");
	brsstrcat((UDINT)&gUdpClient_txbuf[0], (UDINT)"defect_desc_5,");
	brsstrcat((UDINT)&gUdpClient_txbuf[0], (UDINT)"defect_desc_6,");
	brsstrcat((UDINT)&gUdpClient_txbuf[0], (UDINT)"defect_desc_7,");
	brsstrcat((UDINT)&gUdpClient_txbuf[0], (UDINT)"defect_desc_8,");
	brsstrcat((UDINT)&gUdpClient_txbuf[0], (UDINT)"defect_desc_9,");
	brsstrcat((UDINT)&gUdpClient_txbuf[0], (UDINT)"defect_desc_10,");
	brsstrcat((UDINT)&gUdpClient_txbuf[0], (UDINT)"defect_desc_11,");
	brsstrcat((UDINT)&gUdpClient_txbuf[0], (UDINT)"defect_desc_12");
	brsstrcat((UDINT)&gUdpClient_txbuf[0], (UDINT)" FROM ");

	brsstrcat((UDINT)&gUdpClient_txbuf[0], (UDINT)p->activeDBTableName);
	brsstrcat((UDINT)&gUdpClient_txbuf[0], (UDINT)"\"}, \"id\": ");
	brsitoa(p->activeSQLid, (UDINT)textBuf);
	brsstrcat((UDINT)&gUdpClient_txbuf[0], (UDINT)textBuf);
	brsstrcat((UDINT)&gUdpClient_txbuf[0], (UDINT)"}");

	pushSQLQuery(p->activeSQLid, (unsigned char*)gUdpClient_txbuf, brsstrlen((UDINT)gUdpClient_txbuf));
	//gUdpClient.clientIf.iSend = 1;
}

DINT tableFilterGetSelectedItemRawIndexProducts(hmiTableProducts_typ* p, int selectedItem)
{
	DINT ii;
	hmiTableItemDataProduct_typ* pItemsAll;

	if(!p || !p->pItemsAll)
		return 0;

	pItemsAll = (hmiTableItemDataProduct_typ*)p->pItemsAll; //ptr to an array of all records
	//iterate over all records
	for(ii=0; ii<p->itemCountUnfiltered; ii++, pItemsAll++){
		if((pItemsAll->index < 0) || (pItemsAll->index != selectedItem))
			continue;
		return ii;
	}

	return -1;
}

void tableProductsCyclic()
{
	hmiTableProducts_typ* pT = &gHmi.tableViewProducts;

	//table show view
	tableViewShowProducts(pT);

	//table item (row) selection logic
	tableViewItemSelectionProducts(pT);

	//table scroll logic
	tableViewScrollProducts(pT);

	//table filtering (i.e. shift 1 or 2, active or not active)
	tableFilterProducts(pT);
}
//EOF
```

### paiMp.typ - pai Mp types
```iecst
(********************************************************************
 * COPYRIGHT -- pai
 ********************************************************************
 * Package: paiTemplate
 * File: paiMp.typ
 * Author: goran
 * Created: August 28, 2013
 ********************************************************************
 * Data types of package paiMp
 ********************************************************************)
(*########################################################################*)
(*pai specific defines for mapp objects and types*)
(*########################################################################*)

TYPE
	paiFileItemSizeAndDT_typ : 	STRUCT
		strDT : STRING[63];
		strSize : STRING[15];
	END_STRUCT;
	paiMpTemplateFUBs_typ : 	STRUCT
		MpAlarmBasic : MpAlarmBasic;
		MpAlarmBasicUI : MpAlarmBasicUI;
		MpAlarmRegUser : MpAlarmRegUser;
		MpComDump : MpComDump;
		MpComLoggerUI : MpComLoggerUI;
		MpComLinkToParent : MpComLinkToParent;
		MpFileManagerUI : MpFileManagerUI; (*table colum: id-s*)
		MpRecipeRegPar : MpRecipeRegPar;
		MpRecipeRegParSync : MpRecipeRegParSync;
		MpRecipeUI : MpRecipeUI;
		MpRecipeUICustom1 : MpRecipeUI;
		MpRecipeUICustom2 : MpRecipeUI;
		MpRecipeXml : MpRecipeXml;
		MpRecipeXmlCustom1 : MpRecipeXml;
		MpRecipeXmlCustom2 : MpRecipeXml;
	END_STRUCT;
	paiMpTemplateData_typ : 	STRUCT
		MpComIdent : MpComIdentType;
		MpComLoggerUIConnect : MpComLoggerUIConnectType;
		MpRecipeUIConnect : MpRecipeUIConnectType;
		MpRecipeUIConnectCustom1 : MpRecipeUIConnectType;
		MpRecipeUIConnectCustom2 : MpRecipeUIConnectType;
		MpFileManagerUIConnect : MpFileManagerUIConnectType;
		paiFileItemSizeAndDT : ARRAY[0..9]OF paiFileItemSizeAndDT_typ;
	END_STRUCT;
	paiMpTemplate_typ : 	STRUCT
		data : paiMpTemplateData_typ; (*table colum: id-s*)
		fub : paiMpTemplateFUBs_typ;
	END_STRUCT;
END_TYPE
```

### Program Logical/paiComponents/paiPing/paiPingService (ANSIC)

#### paiPingService.var - Local variables
```iecst
(********************************************************************
 * COPYRIGHT --
 ********************************************************************
 * Program: paiPingService
 * File: paiPingService.var
 * Author: goran
 * Created: August 17, 2015
 ********************************************************************
 * Local variables of program paiPingService
 ********************************************************************)
VAR
	gPaiPing : paiPing_typ := (0);
END_VAR
```

### paiConfig.var
```iecst
(********************************************************************
 * COPYRIGHT --
 ********************************************************************
 * Package: ConfigAndRecipes
 * File: ConfigAndRecipes.var
 * Author: goran_2
 * Created: August 06, 2011
 ********************************************************************
 * Variables of package ConfigAndRecipes
 ********************************************************************)
VAR
	gPaiConfigSys : paiConfigSystem_typ := (0); (*Generic System Configruation Data*)
END_VAR
```

- paiCMRightMenuPressed.clm (not shown)

- paiPingStatus.clm (not shown)

- tcpStatus.clm (not shown)

- Header_0.fninfo (not shown)

- Html_SDM.fninfo (not shown)

- MpButton.fninfo (not shown)

- MpBackground.layer (not shown)

- paiMpFileManagerMsgBox.layer (not shown)

- paiMpFileManagerUI.layer (not shown)

- MpNumPad.tpr (not shown)

- NumPad_Limits.tpr (not shown)

### udpApp.typ
```iecst
(********************************************************************
 * COPYRIGHT -- HP
 ********************************************************************
 * File: Global.typ
 * Author: goran
 * Created: January 23, 2013
 ********************************************************************
 * Global data types of project YieldPlus
 ********************************************************************)
(*==========================*)
(*==== UDP Message Header ====*)
(*==========================*)

TYPE
	jsonOverUDPMsgConst_typ :
		( (*Consts used for json messaging over UDP*)
		CONST_JSONMSG_WEIGHTS := 100,
		CONST_JSONMSG_WORKERS := 30,
		CONST_JSONMSG_INSPECTORS := 40,
		CONST_JSONMSG_PRODUCTS := 50,
		CONST_JSONMSG_DASHBMAIN := 60,
		CONST_JSONMSG_WRKTMUPD := 61,
		CONST_JSONMSG_DASHBDEFECTS := 62,
		CONST_JSONMSG_STATIONDATA := 70,
		CONST_JSONMSG_HMISECURITY := 71,
		CONST_JSONMSG_HMILOGGING := 72
		);
	ctrlInterfaceMsgHeader_typ : 	STRUCT
		msgVersion : STRING[31];
		msgCounter : UDINT;
		msgEchoRequest : UDINT;
		msgEchoResponse : UDINT;
	END_STRUCT;
END_TYPE

(*==========================*)
(*==== UDP Message Common===*)
(*==========================*)

TYPE
	ctrlInterfaceCmdScaleCalib_typ : 	STRUCT
		avgBufferSize : UDINT;
		FIRfilter : UDINT;
		mask : UDINT;
		analogConverterSpeed : UDINT;
		calibrationCmd : UDINT; (*Calibration command: 0-normal operation;1-doZero;2-doCalibration*)
		calibrationWt : REAL; (*Calibraton wt*)
	END_STRUCT;
	ctrlInterfaceCmdScaleWt_typ : 	STRUCT
		zeroThresholdWt : REAL; (*threshold wt under which a scale is assumed empty*)
		targetWt : REAL; (*target wt to fill in the infeed bin*)
		weighDelay : REAL; (*delay time to wait wt measurment in order to accept the wt value*)
		zeroDelay : REAL; (*delay time between measuring zero value and pronouncing the zero wt*)
		breakoutTime : REAL; (*time to wait for product to breakaway from the scale. In other words, time to wait for measured weight to drop below zeroThresholdWt*)
		breakoutAttempts : UDINT; (*number of breakout attempts. 0-none (zero the scale) 1..9-try to breakout the product*)
		breakoutMode : UDINT; (*0-rezero scale after breakout time expires, don't stop the machine 1-stop the machine, generate alarm for the user*)
	END_STRUCT;
	ctrlInterfaceCmdRecordOk_typ : 	STRUCT
		lastDBSavedRecId : UDINT; (*record ID of the last successfuly saved data aquisition record*)
	END_STRUCT;
END_TYPE

(*==========================*)
(*==== UDP Command Message ====*)
(*==========================*)

TYPE
	ctrlInterfaceCmd_typ : 	STRUCT
		listQCInspectors : STRING[511];
	END_STRUCT;
END_TYPE
```

### 1stReadme-UDP.txt
```
Package name:
=============
UDP

Desription:
===========
Package contains support for UDP communication.

About:
======
- package consists of two entities:
---paiUDPService: a package that contains support for application independant UDP client and server logic
---appUDP program: a program that implements application specific UDP logic. This program utilizes services provided by the paiUDPService package.
IMPORTANT:
-updserv and udpclient tasks SHOULD be located above the udpApp task in the CPU task list. That way, custom UDP
configuration provided in the init section of the udpApp will have effect.

Dependencies:
=============
- B&R Libraries: AsUDP
- Other: bglib C utilities

Usage:
======
- UDP server configuration: modify code/settings in: paiUDPService/udpserv.c/udpservINIT()
- UDP client configuration: modify code/settings in: paiUDPService/udpclient.c/udpclientINIT()
- for application specific support, add needed code in appUDP (or elsewhere in the program)

Examples:
=============
TODO
```

### paiProjectInfo.typ
```iecst
(********************************************************************
 * COPYRIGHT --
 ********************************************************************
 * Package: paiComponents
 * File: paiBRHW.typ
 * Author: goran
 * Created: June 23, 2015
 ********************************************************************
 * Data types of package paiTelnet
 ********************************************************************)

TYPE
	paiProjectInfo_typ : 	STRUCT
		ProjectDate : STRING[31];
		ProjectVersion : STRING[31];
		ASVersion : STRING[31];
		Company : STRING[79];
		Address : STRING[79];
		CompanyWeb : STRING[79];
		ContactPhone : STRING[79];
		ProjectAbout : STRING[79];
		ProjectInfo : STRING[79];
		ProjectComments : STRING[79];
	END_STRUCT;
END_TYPE
```

### Program Logical/ParameterDownload/CSV_File

#### ExListFile.ab
```automation-basic
FUNCTION_BLOCK ExListFile
;*****************************************************************
;FUB: 			ExFileList
;*****************************************************************
;Discription:
;	This FUB writes the Values from the allocated memory from the FUB
;	CSV-Init in a CSV-File.
;
;Parameter:
;
;Author:	Georg Kreil
;			B&R Eggelsberg
;
;History:	V0.01.1 - 24 June 2003
;					created
;			V0.01.2 - 8 July 2003
;					no changes
;			V0.01.3 - 14 July 2003
;					no changes
;			V0.01.4 - 15 July 2003
;					Error with maximum namelenght corrected
;					displayed strings changed by diplayed year
;					2003 -> 03
;					and without file-extension
;			V0.01.5 - 17 July 2003
;					no changes
;			V0.01.6 - 18 July 2003
;					Possibility to set the focus over a separate value added
;					Output, if it possible to scroll one page up/down  added
;			V0.01.7 - 7 August 2003
;					no changes
;			V0.01.8 - 8 August 2003
;					output strings one charecter shorter
;			V0.01.9 - 11 August 2003
;					no changes
;*****************************************************************

Internal.CRLF[0]= 13
Internal.CRLF[1]= 10
Internal.CRLF[2]= 0

	select Internal.Step

	;*********************************************************************
		state wait
	;*********************************************************************
	;*********************************************************************
	; control memorysize
    when ( (MaxNameLenght+19)*ArrayNum > SizeStringArray) or (MaxNameLenght > 28) do
    	status= MAX_NAMELENGHT_TO_LONG
    	command= 0
	next wait
	;*********************************************************************
	; create file-list
    when (command = FiJOB_CREATE_FILE_LIST ) and (status <> 65535) do
    	status  = 65535
		next file_dir_info
	;*********************************************************************
	; Scroll one line up
    when (command = FiJOB_LIST_UP) and (status <> 65535) do
	    	if(ListboxFocusPos = 0) then
	    		ListboxFocusPos= 0				; set focus
	        	ScrollUp= 0

	    		if (CSV_FileNum = 1) then ; set/reset scrolldown output
		        	ScrollDown= 0
	        	else
		        	ScrollDown= 1
	    		endif

	    	else
	    		ListboxFocusPos= ListboxFocusPos-1			; set focus

	    		if(ListboxFocusPos <> 0)then ;set/reset scrolldown output
		        	ScrollUp= 1
		        else
		        	ScrollUp= 0
		        endif

	    		if (CSV_FileNum = 1) then ; set/reset scrolldown output
		        	ScrollDown= 0
	        	else
		        	ScrollDown= 1
	    		endif

	    		if(Internal.DownLines < NumListboxLines-1)then
	    			Internal.UpLines= Internal.UpLines-1
	    			Internal.DownLines= Internal.DownLines+1
	    		else
	    			Internal.PosFirstLine= Internal.PosFirstLine-1
	    		endif
			endif
		command = 0
		status  = 0
		next wait
	;*********************************************************************
	; Scroll one line down
    when (command = FiJOB_LIST_DOWN) and (status <> 65535) do
	    	if(CSV_FileNum-1 <= ListboxFocusPos) then
	    		ListboxFocusPos= CSV_FileNum-1			; set focus
	    		ScrollDown= 0

	    		if (CSV_FileNum = 1) then ; set/reset scrollup output
		        	ScrollUp= 0
	        	else
		        	ScrollUp= 1
	    		endif

	    	else

	    		ListboxFocusPos= ListboxFocusPos+1			; set focus

	    		if(ListboxFocusPos <> CSV_FileNum-1 )then; set/reset scrollup output
		    		ScrollDown= 1
				else
		    		ScrollDown= 0
				endif

	    		if (CSV_FileNum = 1) then ; set/reset scrollup output
		        	ScrollUp= 0
	        	else
		        	ScrollUp= 1
	    		endif

	    		if(Internal.UpLines < NumListboxLines-1)then
	    			Internal.UpLines= Internal.UpLines+1
	    			Internal.DownLines= Internal.DownLines-1
	    		else
	    			Internal.PosFirstLine= Internal.PosFirstLine+1
	    		endif

			endif
		command = 0
		status  = 0
		next wait
	;*********************************************************************
	; Scroll one page up
    when (command = FiJOB_LIST_PG_UP) and (status <> 65535) do
	        ; there are less files as lines in the listbox
	    	if(ListboxFocusPos <= 0) or (ListboxFocusPos-NumListboxLines = 0)  then
	    		ListboxFocusPos= 0			; set focus
	        	ScrollUp= 0
    			Internal.UpLines= 0
    			Internal.DownLines= NumListboxLines-1
	    		Internal.PosFirstLine= 0

	    		if (CSV_FileNum = 1) then ; set/reset scrolldown output
		        	ScrollDown= 0
	        	else
		        	ScrollDown= 1
	    		endif

			else if ( ListboxFocusPos-NumListboxLines > 30000 )then
	        	ListboxFocusPos= 0			; set focus
	        	ScrollUp= 0
    			Internal.UpLines= 0
    			Internal.DownLines= NumListboxLines-1
	    		Internal.PosFirstLine= 0

	    		if (CSV_FileNum = 1) then ; set/reset scrolldown output
		        	ScrollDown= 0
	        	else
		        	ScrollDown= 1
	    		endif

			else if ( ListboxFocusPos-NumListboxLines > 0 )and ( ListboxFocusPos-NumListboxLines < 30000 )then
	        	ListboxFocusPos= ListboxFocusPos-NumListboxLines			; set focus
	        	ScrollUp= 1

	    		Internal.PosFirstLine= Internal.PosFirstLine - (NumListboxLines -Internal.UpLines)
    			Internal.UpLines= 0
    			Internal.DownLines= NumListboxLines-1

	    		if (CSV_FileNum = 1) then ; set/reset scrolldown output
		        	ScrollDown= 0
	        	else
		        	ScrollDown= 1
	    		endif

			endif
		command = 0
		status  = 0
		next wait
	;*********************************************************************
	; Scroll one page down
    when (command = FiJOB_LIST_PG_DOWN) and (status <> 65535) do
	        ; there are less files as lines in the listbox
	    	if(CSV_FileNum-1 <= ListboxFocusPos+NumListboxLines) then
	    		ListboxFocusPos= CSV_FileNum-1			; set focus
	    		ScrollDown= 0

    			if( CSV_FileNum > NumListboxLines) then
    				Internal.PosFirstLine= (CSV_FileNum-1)-(NumListboxLines-1)
   	 				Internal.UpLines= NumListboxLines-1
    				Internal.DownLines= 0
    			endif

	    		if (CSV_FileNum = 1) then ; set/reset scrollup output
		        	ScrollUp= 0
	        	else
		        	ScrollUp= 1
	    		endif

			else if ( ListboxFocusPos+NumListboxLines > CSV_FileNum )then
	        	ListboxFocusPos= CSV_FileNum-1			; set focus
	    		ScrollDown= 0

    			Internal.PosFirstLine= (CSV_FileNum-1)-(NumListboxLines-1)
    			Internal.UpLines= NumListboxLines-1
    			Internal.DownLines= 0

	    		if (CSV_FileNum = 1) then ; set/reset scrollup output
		        	ScrollUp= 0
	        	else
		        	ScrollUp= 1
	    		endif

			else if ( ListboxFocusPos+NumListboxLines < CSV_FileNum )then
	        	ListboxFocusPos= ListboxFocusPos+NumListboxLines			; set focus
	    		ScrollDown= 1

    			Internal.PosFirstLine= Internal.PosFirstLine + NumListboxLines - Internal.DownLines
    			Internal.UpLines= NumListboxLines-1
    			Internal.DownLines= 0

	    		if (CSV_FileNum = 1) then ; set/reset scrollup output
		        	ScrollUp= 0
	        	else
		        	ScrollUp= 1
	    		endif

			endif
		command = 0
		status  = 0
	    next wait

	;*********************************************************************
	; set focus with input-value
    when (command = FiJOB_SET_FOCUS) and (status <> 65535) do
  		if( SetFocusPos <= NumListboxLines-1  ) then
  			if( CSV_FileNum- 1 >= Internal.PosFirstLine+SetFocusPos ) then
		  		ListboxFocusPos= Internal.PosFirstLine+SetFocusPos
		  		Internal.DownLines= NumListboxLines-SetFocusPos-1
		  		Internal.UpLines= SetFocusPos
				status  = 0
			endif

		else
			status  = FOCUSPOS_OUT_OF_LISTBOX
		endif

	  	command = 0
   		next wait

	;*********************************************************************
		state file_dir_info
	;*********************************************************************

	  ; no memoryadress given
		when ( pStringArray = 0)  do
			command = 0
			status  = ERR_NO_MEM_ALLOC
		next wait

	    DirInfo_CSV.enable = 1
	    DirInfo_CSV.pDevice = pFileDevice
	    DirInfo_CSV.pPath = 0
	    DirInfo_CSV FUB DirInfo()

	    ;no error, files exists
	    when (DirInfo_CSV.status = ERRF_NO_ERROR) and (DirInfo_CSV.filenum <> 0) DO
	      Internal.FileNumOnDisk = uint(DirInfo_CSV.filenum)
	  	  memset(pStringArray, 0, SizeStringArray)
	      CSV_FileNum = 0								; filenumber reset
	      Internal.FileNumAct = 0                      	; actual filenumber reset
	      Internal.Offset = 0							; reset offset
	      status= 65535
		  strcpy(adr(Internal.TmpExtension),".CSV")
	      next file_info

	    ; no error, no files
	    when (DirInfo_CSV.status = ERRF_NO_ERROR) and (DirInfo_CSV.filenum = 0) DO
	      Internal.FileNumOnDisk = 0                    ; number of files reset
	      Internal.FileNumAct = 0                       ; actual filenumber reset
	      CSV_FileNum = 0								; filenumber reset
	   	  memset(pStringArray, 0,SizeStringArray)	  ; clear memory
	      command = 0  	                              ; command reset
	      status= 0  	      						  ; clear status
	      next wait

	    ; Fehler aufgetreten
	    when (DirInfo_CSV.status <> ERRF_NO_ERROR) and (DirInfo_CSV.status <> 65535) DO
	      status = DirInfo_CSV.status                  ; set error
	      command = 0                             	   ; command reset
	      Internal.FileNumAct = 0                      ; actual filenumber reset
	      Internal.Offset = 0      				       ; reset offset
	      next wait

	;*********************************************************************************
	  state file_info
	;*********************************************************************************

	    when (ArrayNum < Internal.FileNumOnDisk) DO
			command = 0
			status  = ARRAY_TO_LESS
    	next wait

	    ; create FileInfo
	    DirRead_CSV.enable = 1
	    DirRead_CSV.pDevice = pFileDevice
	    DirRead_CSV.pPath = 0
	    DirRead_CSV.entry = udint(Internal.FileNumAct)  ; actual filenumber
	    DirRead_CSV.option = FILE_FILE
	    DirRead_CSV.pData = adr(Internal.FileInfo)
	    DirRead_CSV.data_len = sizeof(Internal.FileInfo)
	    DirRead_CSV FUB DirRead()

	    ; Fehler aufgetreten
	    when (DirRead_CSV.status <> 0) and (DirRead_CSV.status <> 65535) do
	      status = DirRead_CSV.status                      ; Fehler setzen
	      command= 0
	      next wait

	    ; no error
	    if (DirRead_CSV.status = 0) then
	      ; filename to long -> not add to filelist
	      if (strlen(adr(Internal.FileInfo.Filename)) <= MaxNameLenght+4) then
			; control, if the file has the right extension
	      	loop Internal.i=0 to strlen(adr(Internal.FileInfo.Filename)) do
		     	memcpy(adr(Internal.TmpExtension),adr(Internal.FileInfo.Filename[Internal.i]),sizeof(Internal.TmpExtension))
		     	Internal.result1=strcmp(adr(Internal.TmpExtension),".CSV")
				Internal.result2=strcmp(adr(Internal.TmpExtension),".csv")

				; File gefunden
				if((Internal.result1 = 0 ) or (Internal.result2 = 0 ))then
					Internal.FileFound = 1
			    else if( adr(Internal.FileInfo.Filename[Internal.i]) = '.' )then
			    	exitif(1=1)			; File hat falsche Extension
			    endif

		    endloop

	      endif

	      Internal.FileNumAct = Internal.FileNumAct + 1                ;  increase actual filenumber
	    endif

		; ein neues CSV-File wurde gefunden
	    when(Internal.FileFound = 1) do
	    	Internal.FileFound = 0
	    	next open_file

	    when (Internal.FileNumAct >= Internal.FileNumOnDisk) DO		; all files listed
			command = 0								; reset command
			ListboxFocusPos= 0						; reset focus-position
	       	ScrollUp= 0
   			Internal.UpLines= 0
   			Internal.DownLines= NumListboxLines-1
   			Internal.PosFirstLine= 0

    		if (CSV_FileNum = 1) then
	        	ScrollDown= 0
        	else
	        	ScrollDown= 1
    		endif

			status  = 0		    					; reset status
      next wait

	;*********************************************************************************
	  state open_file
	;*********************************************************************************

		FileOpen_CSV.enable= 1
		FileOpen_CSV.pDevice= pFileDevice
		FileOpen_CSV.pFile= adr(Internal.FileInfo.Filename)
		FileOpen_CSV.mode= FILE_R
		FileOpen_CSV FUB FileOpen()

			; no error
			when (FileOpen_CSV.status = 0) do
				; allocate memory, to copy the first part of file
				Internal.status_alloc= TMP_alloc(FileOpen_CSV.filelen,adr(Internal.pFileData))
				status= 65535
			next read_file

			; file is opening
			when (FileOpen_CSV.status = 65535) do
				status= FileOpen_CSV.status
			next open_file

			;error durring opening
			when (FileOpen_CSV.status <> 0) and (FileOpen_CSV.status <> 65535) do
				status= FileOpen_CSV.status
			next wait

	;##########################################################################################
	state read_file
	;##########################################################################################

		if( (Internal.status_alloc = 0) and (FileOpen_CSV.status = 0) )then
			FileRead_CSV.enable= 1
			FileRead_CSV.ident= FileOpen_CSV.ident
			FileRead_CSV.offset= 0
			FileRead_CSV.pDest= Internal.pFileData
			FileRead_CSV.len= FileOpen_CSV.filelen
			FileRead_CSV FUB FileRead()
		endif

		; keine Speicher allokiert
		when (Internal.status_alloc <> 0) do
				status= Internal.status_alloc
			next wait

		; Fehler aufgetreten
		when (FileRead_CSV.status <> 0) and  (FileRead_CSV.status <> 65535) do
				status= FileRead_CSV.status
			next wait
		; noch beim Auslesen
		when (FileRead_CSV.status = 65535) do
				status= FileRead_CSV.status
			next read_file

		; fertig mit auslesen
		when (FileRead_CSV.status = 0) do
				status= 65535
			next close_file

		;##########################################################################################
		state close_file
		;##########################################################################################

		 	FileClose_CSV.enable= 1
			FileClose_CSV.ident= FileOpen_CSV.ident
			FileClose_CSV FUB FileClose()

			; Fehler beim Schliessen
			when (FileClose_CSV.status <> 0) and (FileClose_CSV.status <> 65535) do
				status= FileClose_CSV.status
			next wait

			; kein Fehler aufgetreten
			when (FileClose_CSV.status = 0) do
				status= 65535
			next search_filename

			; noch nicht fertig
			when (FileClose_CSV.status = 65535) do
				status= FileClose_CSV.status
			next close_file

		;##########################################################################################
		state search_filename
		;##########################################################################################

		; Kontrolle des Optionspointer
		when pOptions = 0 do
			status = ERR_ZERO_POINTER_OPTION
			next wait

		; Merker zurücksetzen
		Internal.PositionFound = 0
		Internal.FirstSeperatorFound = 0
		Internal.SecondSeperatorFound = 0
		Internal.EndPositionFound = 0

		; Optionsstruktur holen
		; -> kein Zeiger wegen debug-Möglichkeit
		memcpy( adr(Internal.OptionStruct), pOptions, sizeof(Internal.OptionStruct) )

		; ausgelesenes File durchsuchen
      	loop Internal.i=0 to Internal.OptionStruct.FileLenToRead do

      		; Position des Variablennamen im CSV-File suchen
			if (Internal.PositionFound = 0) then
				Internal.result1=memcmp( Internal.pFileData + Internal.i, adr(Internal.OptionStruct.SearchVarName), 5)
				if (Internal.result1 = 0) then
					Internal.PositionFound = 1	; Position gefunden
				endif
			; ersten ';' suchen
			else if (Internal.FirstSeperatorFound = 0 )then
				DynUsint access Internal.pFileData + Internal.i
				if (DynUsint = ';') then
					Internal.FirstSeperatorFound = 1 ; ersten ';' gefunden
				endif
			; zweiten ';' suchen
			else if (Internal.SecondSeperatorFound = 0 )then
				DynUsint access Internal.pFileData + Internal.i
				if (DynUsint = ';') then
					Internal.StartPositionName =  Internal.pFileData + Internal.i + 1 ;Startposition merken
					Internal.SecondSeperatorFound = 1 ; zweiten ';' gefunden
				endif
			; Ende der Zeile suchen
			else if (Internal.EndPositionFound = 0 )then
				DynUsint access Internal.pFileData + Internal.i
				if (DynUsint = 13) then
					; Variablenwert herauskopieren
					memcpy(adr(Internal.InternalFileName), Internal.StartPositionName, Internal.pFileData + Internal.i - Internal.StartPositionName);
					Internal.EndPositionFound = 1 ; Ende der Zeile gefunden
				endif
			endif
		endloop

		; Kompletten String löschen
		memset( adr(Internal.CompleteEntry), 0, sizeof(Internal.CompleteEntry) )
		;echten Filenamen "zusammenstutzen"
		memset( adr(Internal.FileInfo.Filename[strlen(adr(Internal.FileInfo.Filename)) - 4]), 0, sizeof(Internal.FileInfo.Filename)-strlen(adr(Internal.FileInfo.Filename))  )
		if ( strlen(adr(Internal.FileInfo.Filename)) > Internal.OptionStruct.MaxNrLen ) then
			Internal.FileInfo.Filename[Internal.OptionStruct.MaxNrLen] = 0
		else
			loop Internal.i = strlen(adr(Internal.FileInfo.Filename)) to Internal.OptionStruct.MaxNrLen-1 do
				Internal.FileInfo.Filename[Internal.i] = ' '
			endloop
		endif

		;echten Filenamen umkopieren
		memcpy( adr(Internal.CompleteEntry), adr(Internal.FileInfo.Filename) ,strlen(adr(Internal.FileInfo.Filename)) )
;		strcat( adr(Internal.CompleteEntry), "  ")

		;Filenamen "zusammenstutzen"
		if ( strlen(adr(Internal.InternalFileName)) > Internal.OptionStruct.MaxNameLen ) then
			Internal.InternalFileName[Internal.OptionStruct.MaxNameLen] = 0
		else
			loop Internal.i = strlen(adr(Internal.InternalFileName)) to Internal.OptionStruct.MaxNameLen-1 do
				Internal.InternalFileName[Internal.i] = ' '
			endloop
		endif
		;Filenamen hinzufügen zum echten Filenamen
		strcat( adr(Internal.CompleteEntry),adr(Internal.InternalFileName) )

		DT_TO_DTStructure(Internal.FileInfo.Date, adr(Internal.dateandtime));

		; create date and time to a string and add to the filename
		Internal.TmpString[0]= (Internal.dateandtime.day / 10) + '0'
		Internal.TmpString[1]= (Internal.dateandtime.day mod 10) + '0'
		Internal.TmpString[2]= '.'

		Internal.TmpString[3]= (Internal.dateandtime.month / 10) + '0'
		Internal.TmpString[4]= (Internal.dateandtime.month mod 10) + '0'
		Internal.TmpString[5]= '.'

		Internal.TmpString[6]= USINT( ((Internal.dateandtime.year mod 100)/10)  ) + '0'
		Internal.TmpString[7]= USINT(  (Internal.dateandtime.year mod 10)       ) + '0'
		Internal.TmpString[8]= ' '

		Internal.TmpString[9]= (Internal.dateandtime.hour / 10) + '0'
		Internal.TmpString[10]= (Internal.dateandtime.hour mod 10) + '0'
		Internal.TmpString[11]= ':'
		Internal.TmpString[12]= (Internal.dateandtime.minute / 10) + '0'
		Internal.TmpString[13]= (Internal.dateandtime.minute mod 10) + '0'
		Internal.TmpString[14]= 0

;		strcat( adr(Internal.CompleteEntry), " ")
		strcat( adr(Internal.CompleteEntry),adr(Internal.TmpString) )
		memset( adr(Internal.InternalFileName), 0, sizeof(Internal.InternalFileName) )

;		strcpy( pStringArray + Internal.Offset, adr(Internal.CompleteEntry) )
		strcpy( pStringArray + Internal.Offset, adr(Internal.CompleteEntry) )
		Internal.Offset = Internal.Offset + strlen( adr(Internal.CompleteEntry)) + 1

	    inc(CSV_FileNum)				; increase CSV-filenumber

	    when (Internal.FileNumAct >= Internal.FileNumOnDisk) DO		; all files listed
			command = 0								; reset command
			ListboxFocusPos= 0						; reset focus-position
	       	ScrollUp= 0
   			Internal.UpLines= 0
   			Internal.DownLines= NumListboxLines-1
   			Internal.PosFirstLine= 0

    		if (CSV_FileNum = 1) then
	        	ScrollDown= 0
        	else
	        	ScrollDown= 1
    		endif
			status  = 0		    					; reset status
    		next wait

		; nächster File holen
		when (1 = 1) do
			status= 65535
			next file_info

	endselect
END_FUNCTION_BLOCK
```

### P74param.var
```iecst
(********************************************************************
 * COPYRIGHT --
 ********************************************************************
 * Program: P84param
 * File: P84param.var
 * Author: scoccimaroj
 * Created: July 14, 2010
 ********************************************************************
 * Local variables of program P84param
 ********************************************************************)
VAR
	State : USINT;
	cmdStart : BOOL; (*command to start the reading procedure.*)
	eplRead : EplSDORead; (*Function block to read parameters from the drive.*)
	cmdAck : BOOL; (*Acknowledge an epl read error*)
	csvSearch : CSV_Search;
	csvWrite : CSV_WriteFile;
	csvInit : CSV_Init;
	csvInitCheckFile : CSV_InitCheckFile;
	pNames : ARRAY[0..4] OF UDINT;
	csvStrucMem : UDINT;
	csvMemLength : UDINT;
	position : INT;
	i : UINT; (*loop variable*)
END_VAR
```

### Program Logical/ParameterDownload/X64_S44_Download/X64param (IEC) - program that downloads the parameters from the X64 drive.

#### X64paramInit.st
```iecst
(********************************************************************
 * COPYRIGHT --
 ********************************************************************
 * Program: X64param
 * File: X64paramInit.st
 * Author: scoccimaroj
 * Created: July 14, 2010
 ********************************************************************
 * Implementation of program X64param
 ********************************************************************)

PROGRAM _INIT

strcpy( ADR(X64ParRead.pDevice) , ADR('IF5.ST9') );
AsIOAccRead_0.pDeviceName := ADR(X64ParRead.pDevice);
strcpy( ADR(X64ParRead.FileDevice), ADR('CONFIG') );

 (* Initialize the CSV file writing operation *)
 strcpy( ADR(X64ParRead.CsvFileName), ADR(X64ParRead.pDevice) );

 FOR i:= 0 TO 10 BY 1 DO
 	position := FIND(X64ParRead.CsvFileName, '.');

	IF (position <> 0) THEN
 		X64ParRead.CsvFileName := REPLACE(X64ParRead.CsvFileName, '_', 1, position);
	END_IF

 END_FOR

 strcat( ADR(X64ParRead.CsvFileName), ADR('.csv') );

 pNames[0] := ADR('X64ParRead');

 csvInit.pStructName := ADR(pNames);
 csvInit.NumOfStructs := 1;
 csvInit.FullNameLenght := 0;
 csvInit.Options := 0;

 csvInit();

 IF (csvInit.status = 0) THEN
 	csvMemLength := csvInit.MemCounter;
	csvStrucMem := csvInit.pStructMem;

	csvInitCheckFile.MemCounter := csvMemLength;
	csvInitCheckFile.enable := 1;
	csvInitCheckFile();

 END_IF

(* Initialize the parameter channel names *)
strcpy( ADR(X64ParRead.Parameters[0].ChannelName) , ADR('ACC_Input') );
strcpy( ADR(X64ParRead.Parameters[1].ChannelName) , ADR('DEC_Input') );
strcpy( ADR(X64ParRead.Parameters[2].ChannelName) , ADR('LSP_Input') );
strcpy( ADR(X64ParRead.Parameters[3].ChannelName) , ADR('HSP_Input') );
strcpy( ADR(X64ParRead.Parameters[4].ChannelName) , ADR('ITH_Input') );
strcpy( ADR(X64ParRead.Parameters[5].ChannelName) , ADR('UFR_Input') );
strcpy( ADR(X64ParRead.Parameters[6].ChannelName) , ADR('FLG_Input') );
strcpy( ADR(X64ParRead.Parameters[7].ChannelName) , ADR('STA_Input') );
strcpy( ADR(X64ParRead.Parameters[8].ChannelName) , ADR('SLP_Input') );
strcpy( ADR(X64ParRead.Parameters[9].ChannelName) , ADR('JPF_Input') );
strcpy( ADR(X64ParRead.Parameters[10].ChannelName) , ADR('JF2_Input') );
strcpy( ADR(X64ParRead.Parameters[11].ChannelName) , ADR('CLI_Input') );
strcpy( ADR(X64ParRead.Parameters[12].ChannelName) , ADR('TLS_Input') );
strcpy( ADR(X64ParRead.Parameters[13].ChannelName) , ADR('FTD_Input') );
strcpy( ADR(X64ParRead.Parameters[14].ChannelName) , ADR('TTD_Input') );
strcpy( ADR(X64ParRead.Parameters[15].ChannelName) , ADR('CTD_Input') );
strcpy( ADR(X64ParRead.Parameters[16].ChannelName) , ADR('SDS_Input') );
strcpy( ADR(X64ParRead.Parameters[17].ChannelName) , ADR('BFR_Input') );
strcpy( ADR(X64ParRead.Parameters[18].ChannelName) , ADR('UNS_Input') );
strcpy( ADR(X64ParRead.Parameters[19].ChannelName) , ADR('FRS_Input') );
strcpy( ADR(X64ParRead.Parameters[20].ChannelName) , ADR('NCR_Input') );
strcpy( ADR(X64ParRead.Parameters[21].ChannelName) , ADR('NSP_Input') );
strcpy( ADR(X64ParRead.Parameters[22].ChannelName) , ADR('COS_Input') );
strcpy( ADR(X64ParRead.Parameters[23].ChannelName) , ADR('RSC_Input') );
strcpy( ADR(X64ParRead.Parameters[24].ChannelName) , ADR('TUN_Input') );
strcpy( ADR(X64ParRead.Parameters[25].ChannelName) , ADR('UFT_Input') );
strcpy( ADR(X64ParRead.Parameters[26].ChannelName) , ADR('NRD_Input') );
strcpy( ADR(X64ParRead.Parameters[27].ChannelName) , ADR('SFR_Input') );
strcpy( ADR(X64ParRead.Parameters[28].ChannelName) , ADR('TFR_Input') );
strcpy( ADR(X64ParRead.Parameters[29].ChannelName) , ADR('SRF_Input') );
strcpy( ADR(X64ParRead.Parameters[30].ChannelName) , ADR('TCC_Input') );
strcpy( ADR(X64ParRead.Parameters[31].ChannelName) , ADR('TCT_Input') );
strcpy( ADR(X64ParRead.Parameters[32].ChannelName) , ADR('RRS_Input') );
strcpy( ADR(X64ParRead.Parameters[33].ChannelName) , ADR('R2_Input') );
strcpy( ADR(X64ParRead.Parameters[34].ChannelName) , ADR('LAC_Input') );
strcpy( ADR(X64ParRead.Parameters[35].ChannelName) , ADR('FR1_Input') );
strcpy( ADR(X64ParRead.Parameters[36].ChannelName) , ADR('FR2_Input') );
strcpy( ADR(X64ParRead.Parameters[37].ChannelName) , ADR('RFC_Input') );
strcpy( ADR(X64ParRead.Parameters[38].ChannelName) , ADR('CHCF_Input') );
strcpy( ADR(X64ParRead.Parameters[39].ChannelName) , ADR('CD1_Input') );
strcpy( ADR(X64ParRead.Parameters[40].ChannelName) , ADR('CD2_Input') );
strcpy( ADR(X64ParRead.Parameters[41].ChannelName) , ADR('CCS_Input') );
strcpy( ADR(X64ParRead.Parameters[42].ChannelName) , ADR('COP_Input') );
strcpy( ADR(X64ParRead.Parameters[43].ChannelName) , ADR('PST_Input') );
strcpy( ADR(X64ParRead.Parameters[44].ChannelName) , ADR('ROT_Input') );
strcpy( ADR(X64ParRead.Parameters[45].ChannelName) , ADR('RPT_Input') );
strcpy( ADR(X64ParRead.Parameters[46].ChannelName) , ADR('TA1_Input') );
strcpy( ADR(X64ParRead.Parameters[47].ChannelName) , ADR('TA2_Input') );
strcpy( ADR(X64ParRead.Parameters[48].ChannelName) , ADR('TA3_Input') );
strcpy( ADR(X64ParRead.Parameters[49].ChannelName) , ADR('TA4_Input') );
strcpy( ADR(X64ParRead.Parameters[50].ChannelName) , ADR('INR_Input') );
strcpy( ADR(X64ParRead.Parameters[51].ChannelName) , ADR('RPS_Input') );
strcpy( ADR(X64ParRead.Parameters[52].ChannelName) , ADR('FRT_Input') );
strcpy( ADR(X64ParRead.Parameters[53].ChannelName) , ADR('AC2_Input') );
strcpy( ADR(X64ParRead.Parameters[54].ChannelName) , ADR('DE2_Input') );
strcpy( ADR(X64ParRead.Parameters[55].ChannelName) , ADR('BRA_Input') );
strcpy( ADR(X64ParRead.Parameters[56].ChannelName) , ADR('STT_Input') );
strcpy( ADR(X64ParRead.Parameters[57].ChannelName) , ADR('FST_Input') );
strcpy( ADR(X64ParRead.Parameters[58].ChannelName) , ADR('DCF_Input') );
strcpy( ADR(X64ParRead.Parameters[59].ChannelName) , ADR('DCI_Input') );
strcpy( ADR(X64ParRead.Parameters[60].ChannelName) , ADR('IDC_Input') );
strcpy( ADR(X64ParRead.Parameters[61].ChannelName) , ADR('TDC_Input') );
strcpy( ADR(X64ParRead.Parameters[62].ChannelName) , ADR('NST_Input') );
strcpy( ADR(X64ParRead.Parameters[63].ChannelName) , ADR('ADC_Input') );
strcpy( ADR(X64ParRead.Parameters[64].ChannelName) , ADR('TDC1_Input') );
strcpy( ADR(X64ParRead.Parameters[65].ChannelName) , ADR('SDC1_Input') );
strcpy( ADR(X64ParRead.Parameters[66].ChannelName) , ADR('TDC2_Input') );
strcpy( ADR(X64ParRead.Parameters[67].ChannelName) , ADR('SDC2_Input') );
strcpy( ADR(X64ParRead.Parameters[68].ChannelName) , ADR('SA2_Input') );
strcpy( ADR(X64ParRead.Parameters[69].ChannelName) , ADR('SA3_Input') );
strcpy( ADR(X64ParRead.Parameters[70].ChannelName) , ADR('PS2_Input') );
strcpy( ADR(X64ParRead.Parameters[71].ChannelName) , ADR('PS4_Input') );
strcpy( ADR(X64ParRead.Parameters[72].ChannelName) , ADR('PS8_Input') );
strcpy( ADR(X64ParRead.Parameters[73].ChannelName) , ADR('PS16_Input') );
strcpy( ADR(X64ParRead.Parameters[74].ChannelName) , ADR('SP2_Input') );
strcpy( ADR(X64ParRead.Parameters[75].ChannelName) , ADR('SP3_Input') );
strcpy( ADR(X64ParRead.Parameters[76].ChannelName) , ADR('SP4_Input') );
strcpy( ADR(X64ParRead.Parameters[77].ChannelName) , ADR('SP5_Input') );
strcpy( ADR(X64ParRead.Parameters[78].ChannelName) , ADR('SP6_Input') );
strcpy( ADR(X64ParRead.Parameters[79].ChannelName) , ADR('SP7_Input') );
strcpy( ADR(X64ParRead.Parameters[80].ChannelName) , ADR('SP8_Input') );
strcpy( ADR(X64ParRead.Parameters[81].ChannelName) , ADR('SP9_Input') );
strcpy( ADR(X64ParRead.Parameters[82].ChannelName) , ADR('SP10_Input') );
strcpy( ADR(X64ParRead.Parameters[83].ChannelName) , ADR('SP11_Input') );
strcpy( ADR(X64ParRead.Parameters[84].ChannelName) , ADR('SP12_Input') );
strcpy( ADR(X64ParRead.Parameters[85].ChannelName) , ADR('SP13_Input') );
strcpy( ADR(X64ParRead.Parameters[86].ChannelName) , ADR('SP14_Input') );
strcpy( ADR(X64ParRead.Parameters[87].ChannelName) , ADR('SP15_Input') );
strcpy( ADR(X64ParRead.Parameters[88].ChannelName) , ADR('SP16_Input') );
strcpy( ADR(X64ParRead.Parameters[89].ChannelName) , ADR('JOG_Input') );
strcpy( ADR(X64ParRead.Parameters[90].ChannelName) , ADR('JGF_Input') );
strcpy( ADR(X64ParRead.Parameters[91].ChannelName) , ADR('USP_Input') );
strcpy( ADR(X64ParRead.Parameters[92].ChannelName) , ADR('DSP_Input') );
strcpy( ADR(X64ParRead.Parameters[93].ChannelName) , ADR('STR_Input') );
strcpy( ADR(X64ParRead.Parameters[94].ChannelName) , ADR('BLC_Input') );
strcpy( ADR(X64ParRead.Parameters[95].ChannelName) , ADR('BRL_Input') );
strcpy( ADR(X64ParRead.Parameters[96].ChannelName) , ADR('IBR_Input') );
strcpy( ADR(X64ParRead.Parameters[97].ChannelName) , ADR('BRT_Input') );
strcpy( ADR(X64ParRead.Parameters[98].ChannelName) , ADR('BEN_Input') );
strcpy( ADR(X64ParRead.Parameters[99].ChannelName) , ADR('BET_Input') );
strcpy( ADR(X64ParRead.Parameters[100].ChannelName) , ADR('BIP_Input') );
strcpy( ADR(X64ParRead.Parameters[101].ChannelName) , ADR('LC2_Input') );
strcpy( ADR(X64ParRead.Parameters[102].ChannelName) , ADR('CL2_Input') );
strcpy( ADR(X64ParRead.Parameters[103].ChannelName) , ADR('CHP_Input') );
strcpy( ADR(X64ParRead.Parameters[104].ChannelName) , ADR('UNS2_Input') );
strcpy( ADR(X64ParRead.Parameters[105].ChannelName) , ADR('FRS2_Input') );
strcpy( ADR(X64ParRead.Parameters[106].ChannelName) , ADR('NCR2_Input') );
strcpy( ADR(X64ParRead.Parameters[107].ChannelName) , ADR('NSP2_Input') );
strcpy( ADR(X64ParRead.Parameters[108].ChannelName) , ADR('COS2_Input') );
strcpy( ADR(X64ParRead.Parameters[109].ChannelName) , ADR('UFT2_Input') );
strcpy( ADR(X64ParRead.Parameters[110].ChannelName) , ADR('UFR2_Input') );
strcpy( ADR(X64ParRead.Parameters[111].ChannelName) , ADR('FLG2_Input') );
strcpy( ADR(X64ParRead.Parameters[112].ChannelName) , ADR('STA2_Input') );
strcpy( ADR(X64ParRead.Parameters[113].ChannelName) , ADR('SLP2_Input') );
strcpy( ADR(X64ParRead.Parameters[114].ChannelName) , ADR('LAF_Input') );
strcpy( ADR(X64ParRead.Parameters[115].ChannelName) , ADR('LAR_Input') );
strcpy( ADR(X64ParRead.Parameters[116].ChannelName) , ADR('LAS_Input') );
strcpy( ADR(X64ParRead.Parameters[117].ChannelName) , ADR('ATR_Input') );
strcpy( ADR(X64ParRead.Parameters[118].ChannelName) , ADR('TAR_Input') );
strcpy( ADR(X64ParRead.Parameters[119].ChannelName) , ADR('RSF_Input') );
strcpy( ADR(X64ParRead.Parameters[120].ChannelName) , ADR('FLR_Input') );
strcpy( ADR(X64ParRead.Parameters[121].ChannelName) , ADR('ETF_Input') );
strcpy( ADR(X64ParRead.Parameters[122].ChannelName) , ADR('LET_Input') );
strcpy( ADR(X64ParRead.Parameters[123].ChannelName) , ADR('EPL_Input') );
strcpy( ADR(X64ParRead.Parameters[124].ChannelName) , ADR('OPL_Input') );
strcpy( ADR(X64ParRead.Parameters[125].ChannelName) , ADR('IPL_Input') );
strcpy( ADR(X64ParRead.Parameters[126].ChannelName) , ADR('OHL_Input') );
strcpy( ADR(X64ParRead.Parameters[127].ChannelName) , ADR('OLL_Input') );
strcpy( ADR(X64ParRead.Parameters[128].ChannelName) , ADR('COL_Input') );
strcpy( ADR(X64ParRead.Parameters[129].ChannelName) , ADR('TNL_Input') );
strcpy( ADR(X64ParRead.Parameters[130].ChannelName) , ADR('LFF_Input') );
strcpy( ADR(X64ParRead.Parameters[131].ChannelName) , ADR('DRN_Input') );
strcpy( ADR(X64ParRead.Parameters[132].ChannelName) , ADR('STP_Input') );
strcpy( ADR(X64ParRead.Parameters[133].ChannelName) , ADR('INH_Input') );
strcpy( ADR(X64ParRead.Parameters[134].ChannelName) , ADR('FLO_Input') );
strcpy( ADR(X64ParRead.Parameters[135].ChannelName) , ADR('FLOC_Input') );
strcpy( ADR(X64ParRead.Parameters[136].ChannelName) , ADR('COD_Input') );
strcpy( ADR(X64ParRead.Parameters[137].ChannelName) , ADR('DO_Input') );

END_PROGRAM
```

Listed in the project but not available here: Logical/MachineControl/appHmi/appHmiLogic.c, Logical/paiComponents/paiHmi/paiHmiPageChange.c, Logical/paiComponents/paiHmi/paiHmiParamList.c, Logical/paiComponents/bglib/bgstring.c, Logical/paiComponents/bglib/bgBitUtilities.c, Logical/paiComponents/paiHmi/paiHmiDialog.c, Logical/paiComponents/paiFileService/paiFS/paiFile.c, Logical/paiComponents/paiFileService/paiFS/paiFile.h, Logical/paiComponents/bglib/bgstring.c, Logical/paiComponents/paiMp/paiMp.var, Logical/paiComponents/paiMp/paiMp, Logical/paiComponents/paiMp/paiFileDT, Logical/paiComponents/paiPing/paiPingService/paiPingService.c, Logical/paiComponents/paiPing/paiPingService/paiPingService.typ, Logical/paiComponents/paiPing/paiPingService/paiPing.c, Logical/ParameterDownload/P84_Download/P84param, Logical/ParameterDownload/X64_S44_Download/S44param
